(* Enum for exchange the data in FB_CR800Ethercat *)
{attribute 'strict'}
TYPE E_CR800StateCommandExchange :
(
	CR800_CMD_EXCHANGE_IDLE							:= 0,	(*  *)
	CR800_CMD_EXCHANGE_SEND_DATA	 				:= 10,	(*  *)
	CR800_CMD_EXCHANGE_WAIT_FOR_DATA				:= 15,	(*  *)
	CR800_CMD_EXCHANGE_WAIT_FOR_CONFIRMATION 		:= 20,	(*  *)
	CR800_CMD_EXCHANGE_SEND_CONFIRMATION			:= 25,	(*  *)
	CR800_CMD_EXCHANGE_RESET_ITERLOCKS				:= 30,	(*  *)
	CR800_CMD_EXCHANGE_WAIT_FOR_RESET_COMMAND		:= 35,	(*  *)
	CR800_CMD_EXCHANGE_WAIT_FOR_RESET_CONFIRMATION	:= 40,	(*  *)
	CR800_CMD_EXCHANGE_SEND_RESET_CONFIRMATION		:= 45,	(*  *)
	CR800_CMD_EXCHANGE_DONE							:= 50	(*  *)
);
END_TYPE

(* stored: Version 1.1.0.1, ProductVersion 3.1.4024.12
   DUT E_CR800StateCommandExchange: Id {3740e884-63db-441a-b40f-bfd9cb381160} *)
